// TIA Portal V19 export
FUNCTION_BLOCK "Main_Safety_RTG1"   // FB1, F_LAD
{ S7_Optimized_Access := 'TRUE' }
// stored: AutoNumber false
   VAR
      Convoyer7A_Instance : "Convoyer7";
      MainCabinetDiagReset_Instance : "MainCabinetDiagReset";
      Convoyer7B_Instance : "Convoyer7";
   END_VAR
BEGIN

REGION Network 1
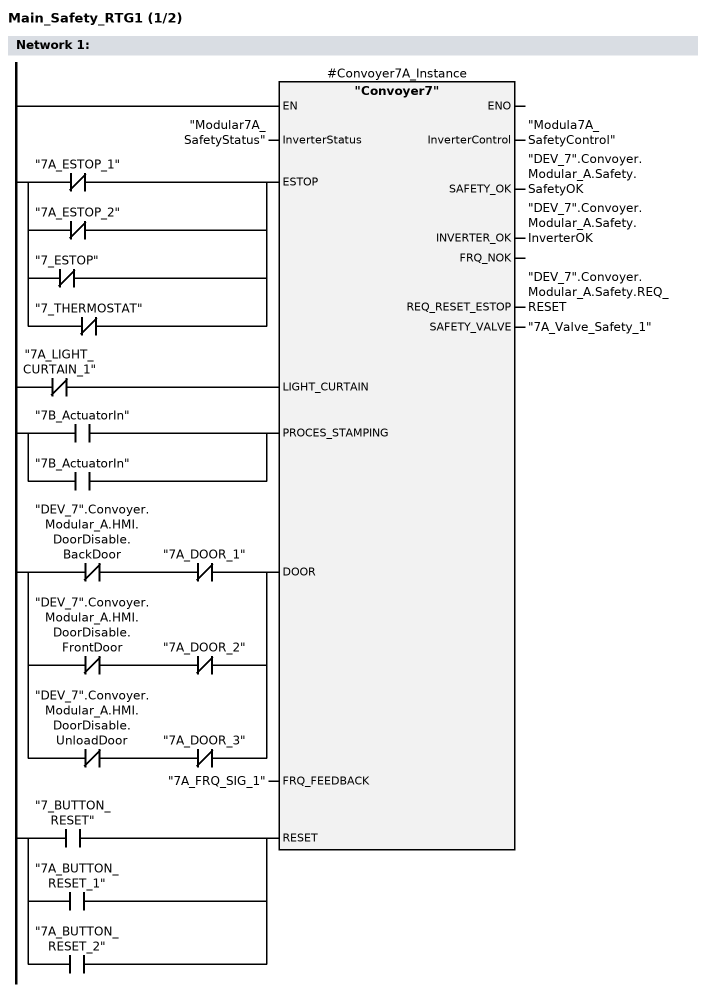
   RUNG wire#powerrail
      #Convoyer7A_Instance(ESTOP := wire#w1, LIGHT_CURTAIN := wire#w2, PROCES_STAMPING := wire#w3, DOOR := wire#w4, RESET := wire#w5, InverterStatus := "Modular7A_SafetyStatus", FRQ_FEEDBACK := "7A_FRQ_SIG_1", InverterControl => "Modula7A_SafetyControl", SAFETY_OK => "DEV_7".Convoyer.Modular_A.Safety.SafetyOK, INVERTER_OK => "DEV_7".Convoyer.Modular_A.Safety.InverterOK, FRQ_NOK =>, REQ_RESET_ESTOP => "DEV_7".Convoyer.Modular_A.Safety.REQ_RESET, SAFETY_VALVE => "7A_Valve_Safety_1")
   END_RUNG
   RUNG wire#powerrail
      I_Contact( "7A_ESTOP_1" )
   END_RUNG wire#w1
   RUNG wire#powerrail
      I_Contact( "7A_ESTOP_2" )
   END_RUNG wire#w1
   RUNG wire#powerrail
      I_Contact( "7_ESTOP" )
   END_RUNG wire#w1
   RUNG wire#powerrail
      I_Contact( "7_THERMOSTAT" )
   END_RUNG wire#w1
   RUNG wire#powerrail
      I_Contact( "7A_LIGHT_CURTAIN_1" )
   END_RUNG wire#w2
   RUNG wire#powerrail
      Contact( "7B_ActuatorIn" )
   END_RUNG wire#w3
   RUNG wire#powerrail
      Contact( "7B_ActuatorIn" )
   END_RUNG wire#w3
   RUNG wire#powerrail
      I_Contact( "DEV_7".Convoyer.Modular_A.HMI.DoorDisable.BackDoor )
      I_Contact( "7A_DOOR_1" )
   END_RUNG wire#w4
   RUNG wire#powerrail
      I_Contact( "DEV_7".Convoyer.Modular_A.HMI.DoorDisable.FrontDoor )
      I_Contact( "7A_DOOR_2" )
   END_RUNG wire#w4
   RUNG wire#powerrail
      I_Contact( "DEV_7".Convoyer.Modular_A.HMI.DoorDisable.UnloadDoor )
      I_Contact( "7A_DOOR_3" )
   END_RUNG wire#w4
   RUNG wire#powerrail
      Contact( "7_BUTTON_RESET" )
   END_RUNG wire#w5
   RUNG wire#powerrail
      Contact( "7A_BUTTON_RESET_1" )
   END_RUNG wire#w5
   RUNG wire#powerrail
      Contact( "7A_BUTTON_RESET_2" )
   END_RUNG wire#w5
   // the same network as SCL:
   #Convoyer7A_Instance(InverterStatus := "Modular7A_SafetyStatus",   // "Convoyer7"
                        ESTOP := NOT "7A_ESTOP_1" OR NOT "7A_ESTOP_2" OR NOT "7_ESTOP" OR NOT "7_THERMOSTAT",
                        LIGHT_CURTAIN := NOT "7A_LIGHT_CURTAIN_1",
                        PROCES_STAMPING := "7B_ActuatorIn" OR "7B_ActuatorIn",
                        DOOR := (NOT "DEV_7".Convoyer.Modular_A.HMI.DoorDisable.BackDoor AND NOT "7A_DOOR_1") OR (NOT "DEV_7".Convoyer.Modular_A.HMI.DoorDisable.FrontDoor AND NOT "7A_DOOR_2") OR (NOT "DEV_7".Convoyer.Modular_A.HMI.DoorDisable.UnloadDoor AND NOT "7A_DOOR_3"),
                        FRQ_FEEDBACK := "7A_FRQ_SIG_1",
                        RESET := "7_BUTTON_RESET" OR "7A_BUTTON_RESET_1" OR "7A_BUTTON_RESET_2",
                        InverterControl => "Modula7A_SafetyControl",
                        SAFETY_OK => "DEV_7".Convoyer.Modular_A.Safety.SafetyOK,
                        INVERTER_OK => "DEV_7".Convoyer.Modular_A.Safety.InverterOK,
                        REQ_RESET_ESTOP => "DEV_7".Convoyer.Modular_A.Safety.REQ_RESET,
                        SAFETY_VALVE => "7A_Valve_Safety_1");
END_REGION

REGION Network 2
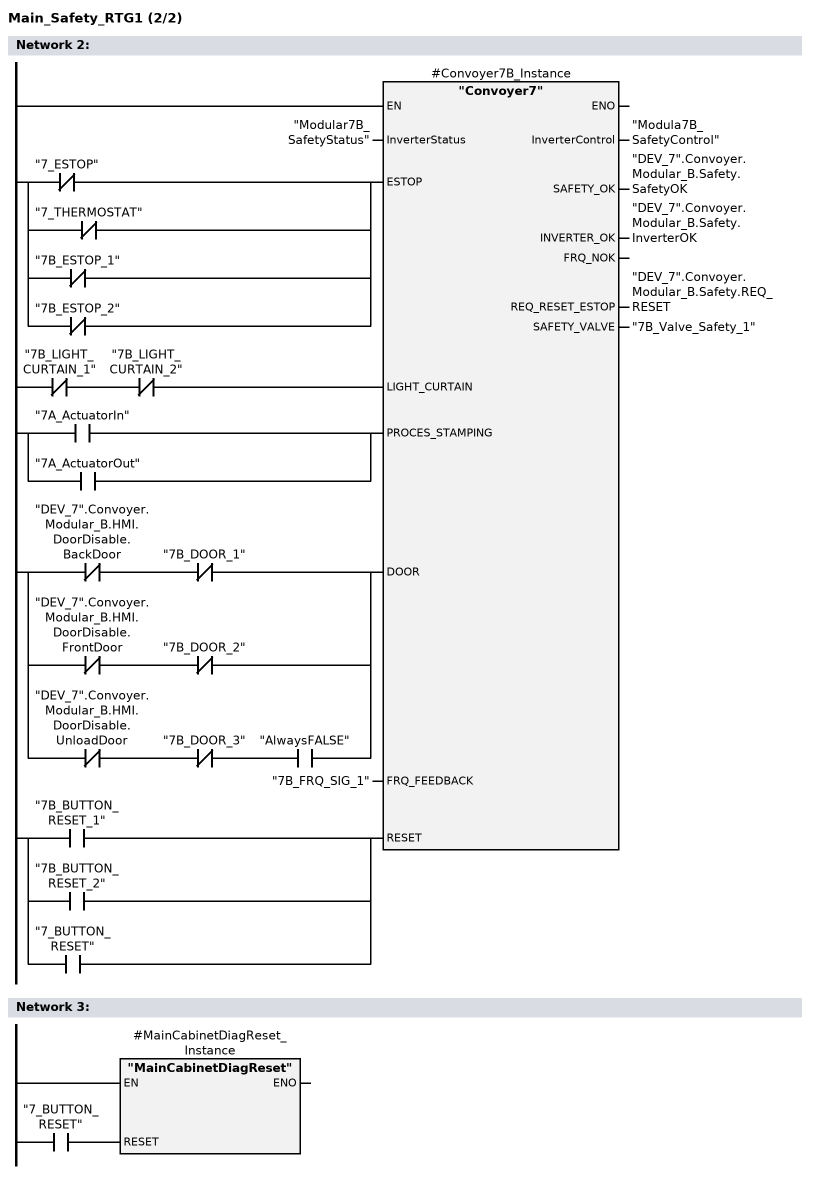
   RUNG wire#powerrail
      #Convoyer7B_Instance(ESTOP := wire#w1, LIGHT_CURTAIN := wire#w2, PROCES_STAMPING := wire#w3, DOOR := wire#w4, RESET := wire#w5, InverterStatus := "Modular7B_SafetyStatus", FRQ_FEEDBACK := "7B_FRQ_SIG_1", InverterControl => "Modula7B_SafetyControl", SAFETY_OK => "DEV_7".Convoyer.Modular_B.Safety.SafetyOK, INVERTER_OK => "DEV_7".Convoyer.Modular_B.Safety.InverterOK, FRQ_NOK =>, REQ_RESET_ESTOP => "DEV_7".Convoyer.Modular_B.Safety.REQ_RESET, SAFETY_VALVE => "7B_Valve_Safety_1")
   END_RUNG
   RUNG wire#powerrail
      I_Contact( "7_ESTOP" )
   END_RUNG wire#w1
   RUNG wire#powerrail
      I_Contact( "7_THERMOSTAT" )
   END_RUNG wire#w1
   RUNG wire#powerrail
      I_Contact( "7B_ESTOP_1" )
   END_RUNG wire#w1
   RUNG wire#powerrail
      I_Contact( "7B_ESTOP_2" )
   END_RUNG wire#w1
   RUNG wire#powerrail
      I_Contact( "7B_LIGHT_CURTAIN_1" )
      I_Contact( "7B_LIGHT_CURTAIN_2" )
   END_RUNG wire#w2
   RUNG wire#powerrail
      Contact( "7A_ActuatorIn" )
   END_RUNG wire#w3
   RUNG wire#powerrail
      Contact( "7A_ActuatorOut" )
   END_RUNG wire#w3
   RUNG wire#powerrail
      I_Contact( "DEV_7".Convoyer.Modular_B.HMI.DoorDisable.BackDoor )
      I_Contact( "7B_DOOR_1" )
   END_RUNG wire#w4
   RUNG wire#powerrail
      I_Contact( "DEV_7".Convoyer.Modular_B.HMI.DoorDisable.FrontDoor )
      I_Contact( "7B_DOOR_2" )
   END_RUNG wire#w4
   RUNG wire#powerrail
      I_Contact( "DEV_7".Convoyer.Modular_B.HMI.DoorDisable.UnloadDoor )
      I_Contact( "7B_DOOR_3" )
      Contact( "AlwaysFALSE" )
   END_RUNG wire#w4
   RUNG wire#powerrail
      Contact( "7B_BUTTON_RESET_1" )
   END_RUNG wire#w5
   RUNG wire#powerrail
      Contact( "7B_BUTTON_RESET_2" )
   END_RUNG wire#w5
   RUNG wire#powerrail
      Contact( "7_BUTTON_RESET" )
   END_RUNG wire#w5
   // the same network as SCL:
   #Convoyer7B_Instance(InverterStatus := "Modular7B_SafetyStatus",   // "Convoyer7"
                        ESTOP := NOT "7_ESTOP" OR NOT "7_THERMOSTAT" OR NOT "7B_ESTOP_1" OR NOT "7B_ESTOP_2",
                        LIGHT_CURTAIN := NOT "7B_LIGHT_CURTAIN_1" AND NOT "7B_LIGHT_CURTAIN_2",
                        PROCES_STAMPING := "7A_ActuatorIn" OR "7A_ActuatorOut",
                        DOOR := (NOT "DEV_7".Convoyer.Modular_B.HMI.DoorDisable.BackDoor AND NOT "7B_DOOR_1") OR (NOT "DEV_7".Convoyer.Modular_B.HMI.DoorDisable.FrontDoor AND NOT "7B_DOOR_2") OR (NOT "DEV_7".Convoyer.Modular_B.HMI.DoorDisable.UnloadDoor AND NOT "7B_DOOR_3" AND "AlwaysFALSE"),
                        FRQ_FEEDBACK := "7B_FRQ_SIG_1",
                        RESET := "7B_BUTTON_RESET_1" OR "7B_BUTTON_RESET_2" OR "7_BUTTON_RESET",
                        InverterControl => "Modula7B_SafetyControl",
                        SAFETY_OK => "DEV_7".Convoyer.Modular_B.Safety.SafetyOK,
                        INVERTER_OK => "DEV_7".Convoyer.Modular_B.Safety.InverterOK,
                        REQ_RESET_ESTOP => "DEV_7".Convoyer.Modular_B.Safety.REQ_RESET,
                        SAFETY_VALVE => "7B_Valve_Safety_1");
END_REGION

REGION Network 3
   RUNG wire#powerrail
      #MainCabinetDiagReset_Instance(RESET := wire#w1)
   END_RUNG
   RUNG wire#powerrail
      Contact( "7_BUTTON_RESET" )
   END_RUNG wire#w1
   // the same network as SCL:
   #MainCabinetDiagReset_Instance(RESET := "7_BUTTON_RESET");   // "MainCabinetDiagReset"
END_REGION
END_FUNCTION_BLOCK
